# B&R Automation Studio project Nikhil_5_Axes
Automation Studio 4.12.2.93; technology packages: mapp 5.24.1, mappCockpit 5.24.1, mappMotion 5.31.0, mappView 5.24.0, mappVision 5.24.0

## Configuration X20CP0484

CPU X20CP0484-1, AutomationRuntime B4.93, Build 4.1.2, Safety 0.0, Vc V4.72.6

### Task classes (Cpu.sw)
```
Cyclic#1 (cycle 4000 us, tolerance 0 us):
  Motion_Con <- Motion_Control.prg
DataObjects: McAcpSys
NcDataObjects: McDriveLog
Binaries: visionUnit, mvLoader, arcoal, arflatprv, arsvcreg, mcprofgen, TCLang, TCData, McPathXT, McAcpSim, mCoWebSc, FWRules, McAcpDrv, udbdef, OpcUaSrv, McMechSys, Role, Config_3, arconfig, Settings, User, asfw, ashwd, Config_1, ashwac, TraceConfi, TC, sysconf, Config_4, Config, Hierarchy, iomap, Config_2, Config_5
Libraries: McBase, MpRobotics, McAxGroup, MpBase, McPathGen, McAxis, McProgInt, McAcpAx, CoTrace, AsZip, FileIO, runtime, ViBase, AsARCfg, powerlnk, AsEPL, AsIO, sys_lib, astime, McStpAx, DataObj, MpAxis, McTrkPath, MpPick, AsOpcUac, AsOpcUas, asarlog, asmem, asieccon, brsystem, asarprof, arssl, asioacc
```

### Hardware
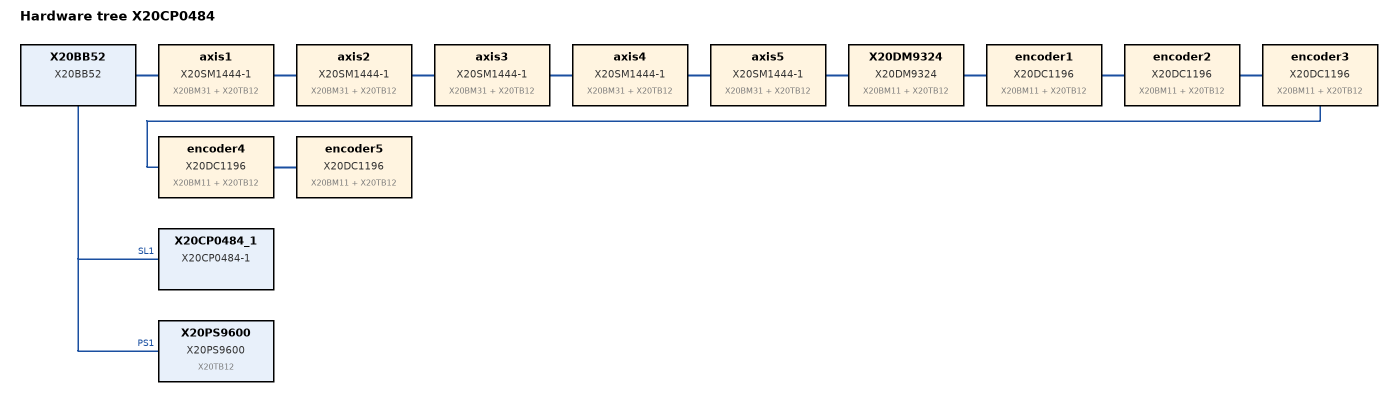
```
X20BB52 : X20BB52 v1.2.0.0
X20BM11 : X20BM11 v1.1.0.0  [X2X1 -> X20BM31d.X2X2]
X20BM11a : X20BM11 v1.1.0.0  [X2X1 -> X20BM11.X2X2]
X20BM11b : X20BM11 v1.1.0.0  [X2X1 -> X20BM11a.X2X2]
X20BM11c : X20BM11 v1.1.0.0  [X2X1 -> X20BM11b.X2X2]
X20BM11d : X20BM11 v1.1.0.0  [X2X1 -> X20BM11c.X2X2]
X20BM11e : X20BM11 v1.1.0.0  [X2X1 -> X20BM11d.X2X2]
X20BM31 : X20BM31 v1.1.0.0  [X2X1 -> X20BB52.IF6]
X20BM31a : X20BM31 v1.1.0.0  [X2X1 -> X20BM31.X2X2]
X20BM31b : X20BM31 v1.1.0.0  [X2X1 -> X20BM31a.X2X2]
X20BM31c : X20BM31 v1.1.0.0  [X2X1 -> X20BM31b.X2X2]
X20BM31d : X20BM31 v1.1.0.0  [X2X1 -> X20BM31c.X2X2]
X20CP0484_1 : X20CP0484-1 v1.4.0.0  [SL -> X20BB52.SL1]
  Connector IF2:
    ActivateDevice = 1
    Mode = Manual
    InternetAddress = 169.254.137.11
    SubnetMask = 255.255.255.0
    InaNodeNumber = 1
    ActivateSnmp = 2
  ConfigurationID = Nikhil_5_Axes
  AutomaticTransferOfUserfiles = on
  MotionLoggerSize = 2048000
  TimerDeviceType = EPLX2X
  TimerDevice = X20BB52.IF6
  TaskClassIdleTime = 4000
  Cyclic1Duration = 4000
  Cyclic1Tolerance = 0
  Cyclic2Duration = 20000
  Cyclic2Tolerance = 20000
  Cyclic3Duration = 48000
  Cyclic3Tolerance = 48000
  Cyclic4Duration = 100000
  Cyclic4Tolerance = 100000
  Cyclic5Duration = 200000
  Cyclic5Tolerance = 200000
  Cyclic6Duration = 500000
  Cyclic6Tolerance = 500000
  Cyclic7Duration = 1000000
  Cyclic7Tolerance = 1000000
  Cyclic8Duration = 8000
  Cyclic8Tolerance = 30000000
  FileDevice1
  FileDeviceName1 = Simulation
  FileDevicePath1 = Z:\Nikhil\Project_5_Axes\Nikhil_test\Logical\CNC_PrgDir
  FileDevice2
  FileDeviceName2 = CNC_PrgDir
  FileDevicePath2 = F:\
  FileDevice3
  FileDeviceName3 = SceneViewer
  FileDevicePath3 = Z:\Nikhil\Project_5_Axes\Nikhil_test\Logical\SceneViewer
  ActivateDns = 1
  DnsDefaultDomain = br-automation.co.at
  FtpUser1
  FtpUsername1 = user
  FtpUserPassword1 = soUu8fSmbl9vOUGFZLohNxYIHTvfYbNb9FbAKhZ+648=
  FtpUserSalt1 = plFIy1g6
  FTPAccessRight1 = 0
  FTPdevice1 = ALL
  ActivateDtmServer = 1
  ActivateOpcUa = 1
  OpcUaPort = 48400
  OpcUa_AuthenticationSecurityPolicy_EnableNone = 1
  OpcUa_AuthenticationSecurityPolicy_EnableBasic128Rsa15 = 1
  OpcUa_Security_AdminRole = Administrators
  OpcUa_Security_EngineerRole = Everyone
  OpcUa_Security_ObserverRole = Everyone
  OpcUaInformationModels_PV_Version = 2
  OpcUaInformationModel_Facet = 0
  OpcUaInformationModel_TypeInformation = 0
  OpcUaInformationModel_BaseObjectTypeForStructures = 0
X20DM9324 : X20DM9324 v1.2.0.0  [SS1 -> X20TB12f.SS; SL -> X20BM11.SL1]
X20PS9600 : X20PS9600 v1.6.0.0  [PS -> X20BB52.PS1; SS1 -> X20TB12.SS]
X20TB12 : X20TB12 v1.0.0.0
X20TB12a : X20TB12 v1.0.0.0
X20TB12b : X20TB12 v1.0.0.0
X20TB12c : X20TB12 v1.0.0.0
X20TB12d : X20TB12 v1.0.0.0
X20TB12e : X20TB12 v1.0.0.0
X20TB12f : X20TB12 v1.0.0.0
X20TB12g : X20TB12 v1.0.0.0
X20TB12h : X20TB12 v1.0.0.0
X20TB12i : X20TB12 v1.0.0.0
X20TB12j : X20TB12 v1.0.0.0
X20TB12k : X20TB12 v1.0.0.0
axis1 : X20SM1444-1 v1.2.0.0  [SS1 -> X20TB12a.SS; SL -> X20BM31.SL1]
  FunctionModel/DriveConfiguration/Module:
    ActivateModuleSimulationOnPLC = Off
  FunctionModel/DriveConfiguration:
    ModuleParameters = StepperParameters
  FunctionModel/DriveConfiguration/ModuleParameters:
    McStepperTypeID = X20Config
    EncoderType = IncrementalDiff
    ReferencePulse = yes
    RatedCurrent = 5.0
    MaximumCurrent = 10.0
    AxesNumber = 1
    FullStepThreshold = 1
    StallDetection = 2
    SmartCurrentControl = 1
    BrakeOutput = 0
    NumberOfDigitalInputs = 3
    NumberOfTriggers = 1
  FunctionModel/DriveConfiguration/Channel[1]/RealAxis:
    AxisReference = gAxisQ1
  FunctionModel/DriveConfiguration/Channel[1]/RealAxis/MechanicalElements/Gearbox:
    InputIsReadOnly = 0
    Input = 48
    OutputIsReadOnly = 0
    Output = 1
  FunctionModel/DriveConfiguration/Channel[1]/RealAxis/MechanicalElements/RotaryToLinearTransformation:
    ReferenceDistanceIsReadOnly = 0
    ReferenceDistance = 1
  FunctionModel/DriveConfiguration/Channel[1]/RealAxis/Motor:
    SteppingAngle = 1.8
  FunctionModel/DriveConfiguration/Channel[1]/RealAxis:
    EncoderLink = OneEncoder
  FunctionModel/DriveConfiguration/Channel[1]/RealAxis/EncoderLink:
    PositionEncoder = External
  FunctionModel/DriveConfiguration/Channel[1]/RealAxis/EncoderLink/PositionEncoder:
    LinesPerRevolution = 2000
    PositionType = Incremental
  FunctionModel/DriveConfiguration/Channel[1]/RealAxis/EncoderLink/PositionEncoder/PositionSource:
    ChannelMapping = %ID.IF6.ST7.Encoder01
  FunctionModel/DriveConfiguration/Channel[1]/RealAxis/EncoderLink/PositionEncoder/ValidityCheck:
    ModuleOk = IOChannel
  FunctionModel/DriveConfiguration/Channel[1]/RealAxis/EncoderLink/PositionEncoder/ValidityCheck/ModuleOk:
    ChannelMapping = %IX.IF6.ST7.ModuleOk
  FunctionModel/DriveConfiguration/Channel[1]/RealAxis/EncoderLink/PositionEncoder/ValidityCheck:
    StaleData = IOChannel
  FunctionModel/DriveConfiguration/Channel[1]/RealAxis/EncoderLink/PositionEncoder/ValidityCheck/StaleData:
    ChannelMapping = %IX.IF6.ST7.StaleData
  FunctionModel/DriveConfiguration/Channel[1]/RealAxis/EncoderLink/PositionEncoder:
    ReferencePulse = NotUsed
  FunctionModel/DriveConfiguration/Channel[1]/RealAxis/EncoderLink/PositionEncoder/PositionFilter:
    PositionFilterTimeConstant = 0.0
    ExtrapolationTime = 0.0
  FunctionModel/DriveConfiguration/Channel[1]/RealAxis/Controller:
    ModeIsReadOnly = 0
    Mode = CurrentController
  FunctionModel/DriveConfiguration/Channel[1]/RealAxis/Controller/Mode/Current:
    StandstillCurrent = 1
    ConstantSpeedCurrent = 4
    SpeedChangeCurrent = 4.2
    FullStepThreshold = 0.0
    MotorSettlingTime = 1
    DelayedCurrentSwitchOff = 1
  FunctionModel/DriveConfiguration/Channel[1]/RealAxis/Homing:
    Mode = AbsoluteSwitch
  FunctionModel/DriveConfiguration/Channel[1]/RealAxis/Homing/Mode:
    Position = 0.0
    StartVelocity = 5.0
    HomingVelocity = 2
    Acceleration = 50.0
    SwitchEdge = Positive
    HomingDirection = Positive
    KeepDirection = No
    ReferencePulse = NotUsed
  FunctionModel/DriveConfiguration/Channel[1]/RealAxis/Homing:
    RestorePositionVariable = 
    ClearPositionError = No
  FunctionModel/DriveConfiguration/Channel[1]/RealAxis/StopReaction:
    DriveError = DecelerationLimit
  FunctionModel/DriveConfiguration/Channel[1]/RealAxis/MovementErrorLimits:
    PositionError = 1000
    StallguardConfiguration = NotUsed
  FunctionModel/DriveConfiguration/Channel[1]/RealAxis:
    JerkFilter = NotUsed
    ZeroVibrationFilter = NotUsed
  FunctionModel/DriveConfiguration/Channel[1]/RealAxis/DigitalInputs/HomingSwitch:
    Source = IOChannel
  FunctionModel/DriveConfiguration/Channel[1]/RealAxis/DigitalInputs/HomingSwitch/Source:
    ChannelMapping = %IX.IF6.ST6.DigitalInput01
  FunctionModel/DriveConfiguration/Channel[1]/RealAxis/DigitalInputs/HomingSwitch:
    Level = Low
  FunctionModel/DriveConfiguration/Channel[1]/RealAxis/DigitalInputs/PositiveLimitSwitch:
    Source = NotUsed
    Level = High
  FunctionModel/DriveConfiguration/Channel[1]/RealAxis/DigitalInputs/NegativeLimitSwitch:
    Source = NotUsed
    Level = High
  FunctionModel/DriveConfiguration/Channel[1]/RealAxis/DigitalInputs/Trigger1:
    Source = NotUsed
    Level = High
  FunctionModel/DriveConfiguration/Channel[1]/RealAxis/DigitalInputs/Trigger2:
    Source = NotUsed
    Level = High
  FunctionModel/DriveConfiguration/Channel[1]/RealAxis/DigitalInputs/Quickstop:
    Input = NotUsed
  FunctionModel/DriveConfiguration/Channel[1]/RealAxis/DigitalOutputs:
    BrakeControl = NotUsed
  FunctionModel/DriveConfiguration/Channel[1]/RealAxis/Simulation:
    LoadSimulationMode = NotUsed
axis2 : X20SM1444-1 v1.2.0.0  [SS1 -> X20TB12b.SS; SL -> X20BM31a.SL1]
  FunctionModel/DriveConfiguration/Module:
    ActivateModuleSimulationOnPLC = Off
  FunctionModel/DriveConfiguration:
    ModuleParameters = StepperParameters
  FunctionModel/DriveConfiguration/ModuleParameters:
    McStepperTypeID = X20Config
    EncoderType = IncrementalDiff
    ReferencePulse = yes
    RatedCurrent = 5.0
    MaximumCurrent = 10.0
    AxesNumber = 1
    FullStepThreshold = 1
    StallDetection = 2
    SmartCurrentControl = 1
    BrakeOutput = 0
    NumberOfDigitalInputs = 3
    NumberOfTriggers = 1
  FunctionModel/DriveConfiguration/Channel[1]/RealAxis:
    AxisReference = gAxisQ2
  FunctionModel/DriveConfiguration/Channel[1]/RealAxis/MechanicalElements/Gearbox:
    InputIsReadOnly = 0
    Input = 48
    OutputIsReadOnly = 0
    Output = 1
  FunctionModel/DriveConfiguration/Channel[1]/RealAxis/MechanicalElements/RotaryToLinearTransformation:
    ReferenceDistanceIsReadOnly = 0
    ReferenceDistance = 1
  FunctionModel/DriveConfiguration/Channel[1]/RealAxis/Motor:
    SteppingAngle = 1.8
  FunctionModel/DriveConfiguration/Channel[1]/RealAxis:
    EncoderLink = OneEncoder
  FunctionModel/DriveConfiguration/Channel[1]/RealAxis/EncoderLink:
    PositionEncoder = External
  FunctionModel/DriveConfiguration/Channel[1]/RealAxis/EncoderLink/PositionEncoder:
    LinesPerRevolution = 2000
    PositionType = Incremental
  FunctionModel/DriveConfiguration/Channel[1]/RealAxis/EncoderLink/PositionEncoder/PositionSource:
    ChannelMapping = %ID.IF6.ST8.Encoder01
  FunctionModel/DriveConfiguration/Channel[1]/RealAxis/EncoderLink/PositionEncoder/ValidityCheck:
    ModuleOk = IOChannel
  FunctionModel/DriveConfiguration/Channel[1]/RealAxis/EncoderLink/PositionEncoder/ValidityCheck/ModuleOk:
    ChannelMapping = %IX.IF6.ST8.ModuleOk
  FunctionModel/DriveConfiguration/Channel[1]/RealAxis/EncoderLink/PositionEncoder/ValidityCheck:
    StaleData = IOChannel
  FunctionModel/DriveConfiguration/Channel[1]/RealAxis/EncoderLink/PositionEncoder/ValidityCheck/StaleData:
    ChannelMapping = %IX.IF6.ST8.StaleData
  FunctionModel/DriveConfiguration/Channel[1]/RealAxis/EncoderLink/PositionEncoder:
    ReferencePulse = NotUsed
  FunctionModel/DriveConfiguration/Channel[1]/RealAxis/EncoderLink/PositionEncoder/PositionFilter:
    PositionFilterTimeConstant = 0.0
    ExtrapolationTime = 0.0
  FunctionModel/DriveConfiguration/Channel[1]/RealAxis/Controller:
    ModeIsReadOnly = 0
    Mode = CurrentController
  FunctionModel/DriveConfiguration/Channel[1]/RealAxis/Controller/Mode/Current:
    StandstillCurrent = 1
    ConstantSpeedCurrent = 4.2
    SpeedChangeCurrent = 4.2
    FullStepThreshold = 0.0
    MotorSettlingTime = 1
    DelayedCurrentSwitchOff = 1
  FunctionModel/DriveConfiguration/Channel[1]/RealAxis/Homing:
    Mode = AbsoluteSwitch
  FunctionModel/DriveConfiguration/Channel[1]/RealAxis/Homing/Mode:
    Position = -10
    StartVelocity = 5.0
    HomingVelocity = 2
    Acceleration = 50.0
    SwitchEdge = Negative
    HomingDirection = Negative
    KeepDirection = No
    ReferencePulse = NotUsed
  FunctionModel/DriveConfiguration/Channel[1]/RealAxis/Homing:
    RestorePositionVariable = 
    ClearPositionError = No
  FunctionModel/DriveConfiguration/Channel[1]/RealAxis/StopReaction:
    DriveError = DecelerationLimit
  FunctionModel/DriveConfiguration/Channel[1]/RealAxis/MovementErrorLimits:
    PositionError = 1000
    StallguardConfiguration = NotUsed
  FunctionModel/DriveConfiguration/Channel[1]/RealAxis:
    JerkFilter = NotUsed
    ZeroVibrationFilter = NotUsed
  FunctionModel/DriveConfiguration/Channel[1]/RealAxis/DigitalInputs/HomingSwitch:
    Source = IOChannel
  FunctionModel/DriveConfiguration/Channel[1]/RealAxis/DigitalInputs/HomingSwitch/Source:
    ChannelMapping = %IX.IF6.ST6.DigitalInput02
  FunctionModel/DriveConfiguration/Channel[1]/RealAxis/DigitalInputs/HomingSwitch:
    Level = Low
  FunctionModel/DriveConfiguration/Channel[1]/RealAxis/DigitalInputs/PositiveLimitSwitch:
    Source = NotUsed
    Level = High
  FunctionModel/DriveConfiguration/Channel[1]/RealAxis/DigitalInputs/NegativeLimitSwitch:
    Source = NotUsed
    Level = High
  FunctionModel/DriveConfiguration/Channel[1]/RealAxis/DigitalInputs/Trigger1:
    Source = NotUsed
    Level = High
  FunctionModel/DriveConfiguration/Channel[1]/RealAxis/DigitalInputs/Trigger2:
    Source = NotUsed
    Level = High
  FunctionModel/DriveConfiguration/Channel[1]/RealAxis/DigitalInputs/Quickstop:
    Input = NotUsed
  FunctionModel/DriveConfiguration/Channel[1]/RealAxis/DigitalOutputs:
    BrakeControl = NotUsed
  FunctionModel/DriveConfiguration/Channel[1]/RealAxis/Simulation:
    LoadSimulationMode = NotUsed
axis3 : X20SM1444-1 v1.2.0.0  [SS1 -> X20TB12c.SS; SL -> X20BM31b.SL1]
  FunctionModel/DriveConfiguration/Module:
    ActivateModuleSimulationOnPLC = Off
  FunctionModel/DriveConfiguration:
    ModuleParameters = StepperParameters
  FunctionModel/DriveConfiguration/ModuleParameters:
    McStepperTypeID = X20Config
    EncoderType = IncrementalDiff
    ReferencePulse = yes
    RatedCurrent = 5.0
    MaximumCurrent = 10.0
    AxesNumber = 1
    FullStepThreshold = 1
    StallDetection = 2
    SmartCurrentControl = 1
    BrakeOutput = 0
    NumberOfDigitalInputs = 3
    NumberOfTriggers = 1
  FunctionModel/DriveConfiguration/Channel[1]/RealAxis:
    AxisReference = gAxisQ3
  FunctionModel/DriveConfiguration/Channel[1]/RealAxis/MechanicalElements/Gearbox:
    InputIsReadOnly = 0
    Input = 50
    OutputIsReadOnly = 0
    Output = 1
  FunctionModel/DriveConfiguration/Channel[1]/RealAxis/MechanicalElements/RotaryToLinearTransformation:
    ReferenceDistanceIsReadOnly = 0
    ReferenceDistance = 1
  FunctionModel/DriveConfiguration/Channel[1]/RealAxis/Motor:
    SteppingAngle = 1.8
  FunctionModel/DriveConfiguration/Channel[1]/RealAxis:
    EncoderLink = OneEncoder
  FunctionModel/DriveConfiguration/Channel[1]/RealAxis/EncoderLink:
    PositionEncoder = External
  FunctionModel/DriveConfiguration/Channel[1]/RealAxis/EncoderLink/PositionEncoder:
    LinesPerRevolution = 2000
    PositionType = Incremental
  FunctionModel/DriveConfiguration/Channel[1]/RealAxis/EncoderLink/PositionEncoder/PositionSource:
    ChannelMapping = %ID.IF6.ST9.Encoder01
  FunctionModel/DriveConfiguration/Channel[1]/RealAxis/EncoderLink/PositionEncoder/ValidityCheck:
    ModuleOk = IOChannel
  FunctionModel/DriveConfiguration/Channel[1]/RealAxis/EncoderLink/PositionEncoder/ValidityCheck/ModuleOk:
    ChannelMapping = %IX.IF6.ST9.ModuleOk
  FunctionModel/DriveConfiguration/Channel[1]/RealAxis/EncoderLink/PositionEncoder/ValidityCheck:
    StaleData = IOChannel
  FunctionModel/DriveConfiguration/Channel[1]/RealAxis/EncoderLink/PositionEncoder/ValidityCheck/StaleData:
    ChannelMapping = %IX.IF6.ST9.StaleData
  FunctionModel/DriveConfiguration/Channel[1]/RealAxis/EncoderLink/PositionEncoder:
    ReferencePulse = NotUsed
  FunctionModel/DriveConfiguration/Channel[1]/RealAxis/EncoderLink/PositionEncoder/PositionFilter:
    PositionFilterTimeConstant = 0.0
    ExtrapolationTime = 0.0
  FunctionModel/DriveConfiguration/Channel[1]/RealAxis/Controller:
    ModeIsReadOnly = 0
    Mode = CurrentController
  FunctionModel/DriveConfiguration/Channel[1]/RealAxis/Controller/Mode/Current:
    StandstillCurrent = 1
    ConstantSpeedCurrent = 4.2
    SpeedChangeCurrent = 4.2
    FullStepThreshold = 0.0
    MotorSettlingTime = 1
    DelayedCurrentSwitchOff = 1
  FunctionModel/DriveConfiguration/Channel[1]/RealAxis/Homing:
    Mode = AbsoluteSwitch
  FunctionModel/DriveConfiguration/Channel[1]/RealAxis/Homing/Mode:
    Position = 10
    StartVelocity = 5.0
    HomingVelocity = 2
    Acceleration = 50.0
    SwitchEdge = Negative
    HomingDirection = Negative
    KeepDirection = No
    ReferencePulse = NotUsed
  FunctionModel/DriveConfiguration/Channel[1]/RealAxis/Homing:
    RestorePositionVariable = 
    ClearPositionError = No
  FunctionModel/DriveConfiguration/Channel[1]/RealAxis/StopReaction:
    DriveError = DecelerationLimit
  FunctionModel/DriveConfiguration/Channel[1]/RealAxis/MovementErrorLimits:
    PositionError = 1000
    StallguardConfiguration = NotUsed
  FunctionModel/DriveConfiguration/Channel[1]/RealAxis:
    JerkFilter = NotUsed
    ZeroVibrationFilter = NotUsed
  FunctionModel/DriveConfiguration/Channel[1]/RealAxis/DigitalInputs/HomingSwitch:
    Source = IOChannel
  FunctionModel/DriveConfiguration/Channel[1]/RealAxis/DigitalInputs/HomingSwitch/Source:
    ChannelMapping = %IX.IF6.ST6.DigitalInput03
  FunctionModel/DriveConfiguration/Channel[1]/RealAxis/DigitalInputs/HomingSwitch:
    Level = Low
  FunctionModel/DriveConfiguration/Channel[1]/RealAxis/DigitalInputs/PositiveLimitSwitch:
    Source = NotUsed
    Level = High
  FunctionModel/DriveConfiguration/Channel[1]/RealAxis/DigitalInputs/NegativeLimitSwitch:
    Source = NotUsed
    Level = High
  FunctionModel/DriveConfiguration/Channel[1]/RealAxis/DigitalInputs/Trigger1:
    Source = NotUsed
    Level = High
  FunctionModel/DriveConfiguration/Channel[1]/RealAxis/DigitalInputs/Trigger2:
    Source = NotUsed
    Level = High
  FunctionModel/DriveConfiguration/Channel[1]/RealAxis/DigitalInputs/Quickstop:
    Input = NotUsed
  FunctionModel/DriveConfiguration/Channel[1]/RealAxis/DigitalOutputs:
    BrakeControl = NotUsed
  FunctionModel/DriveConfiguration/Channel[1]/RealAxis/Simulation:
    LoadSimulationMode = NotUsed
axis4 : X20SM1444-1 v1.2.0.0  [SS1 -> X20TB12d.SS; SL -> X20BM31c.SL1]
  FunctionModel/DriveConfiguration/Module:
    ActivateModuleSimulationOnPLC = Off
  FunctionModel/DriveConfiguration:
    ModuleParameters = StepperParameters
  FunctionModel/DriveConfiguration/ModuleParameters:
    McStepperTypeID = X20Config
    EncoderType = IncrementalDiff
    ReferencePulse = yes
    RatedCurrent = 5.0
    MaximumCurrent = 10.0
    AxesNumber = 1
    FullStepThreshold = 1
    StallDetection = 2
    SmartCurrentControl = 1
    BrakeOutput = 0
    NumberOfDigitalInputs = 3
    NumberOfTriggers = 1
  FunctionModel/DriveConfiguration/Channel[1]/RealAxis:
    AxisReference = gAxisQ4
  FunctionModel/DriveConfiguration/Channel[1]/RealAxis/MechanicalElements/Gearbox:
    InputIsReadOnly = 0
    Input = 40
    OutputIsReadOnly = 0
    Output = 1
  FunctionModel/DriveConfiguration/Channel[1]/RealAxis/MechanicalElements/RotaryToLinearTransformation:
    ReferenceDistanceIsReadOnly = 0
    ReferenceDistance = 1
  FunctionModel/DriveConfiguration/Channel[1]/RealAxis/Motor:
    SteppingAngle = 1.8
  FunctionModel/DriveConfiguration/Channel[1]/RealAxis:
    EncoderLink = OneEncoder
  FunctionModel/DriveConfiguration/Channel[1]/RealAxis/EncoderLink:
    PositionEncoder = External
  FunctionModel/DriveConfiguration/Channel[1]/RealAxis/EncoderLink/PositionEncoder:
    LinesPerRevolution = 2000
    PositionType = Incremental
  FunctionModel/DriveConfiguration/Channel[1]/RealAxis/EncoderLink/PositionEncoder/PositionSource:
    ChannelMapping = %ID.IF6.ST10.Encoder01
  FunctionModel/DriveConfiguration/Channel[1]/RealAxis/EncoderLink/PositionEncoder/ValidityCheck:
    ModuleOk = IOChannel
  FunctionModel/DriveConfiguration/Channel[1]/RealAxis/EncoderLink/PositionEncoder/ValidityCheck/ModuleOk:
    ChannelMapping = %IX.IF6.ST10.ModuleOk
  FunctionModel/DriveConfiguration/Channel[1]/RealAxis/EncoderLink/PositionEncoder/ValidityCheck:
    StaleData = IOChannel
  FunctionModel/DriveConfiguration/Channel[1]/RealAxis/EncoderLink/PositionEncoder/ValidityCheck/StaleData:
    ChannelMapping = %IX.IF6.ST10.StaleData
  FunctionModel/DriveConfiguration/Channel[1]/RealAxis/EncoderLink/PositionEncoder:
    ReferencePulse = NotUsed
  FunctionModel/DriveConfiguration/Channel[1]/RealAxis/EncoderLink/PositionEncoder/PositionFilter:
    PositionFilterTimeConstant = 0.0
    ExtrapolationTime = 0.0
  FunctionModel/DriveConfiguration/Channel[1]/RealAxis/Controller:
    ModeIsReadOnly = 0
    Mode = CurrentController
  FunctionModel/DriveConfiguration/Channel[1]/RealAxis/Controller/Mode/Current:
    StandstillCurrent = 0.6
    ConstantSpeedCurrent = 1.8
    SpeedChangeCurrent = 1.8
    FullStepThreshold = 0.0
    MotorSettlingTime = 1
    DelayedCurrentSwitchOff = 1
  FunctionModel/DriveConfiguration/Channel[1]/RealAxis/Homing:
    Mode = AbsoluteSwitch
  FunctionModel/DriveConfiguration/Channel[1]/RealAxis/Homing/Mode:
    Position = -10
    StartVelocity = 5.0
    HomingVelocity = 2
    Acceleration = 50.0
    SwitchEdge = Positive
    HomingDirection = Positive
    KeepDirection = No
    ReferencePulse = NotUsed
  FunctionModel/DriveConfiguration/Channel[1]/RealAxis/Homing:
    RestorePositionVariable = 
    ClearPositionError = No
  FunctionModel/DriveConfiguration/Channel[1]/RealAxis/StopReaction:
    DriveError = DecelerationLimit
  FunctionModel/DriveConfiguration/Channel[1]/RealAxis/MovementErrorLimits:
    PositionError = 1000
    StallguardConfiguration = NotUsed
  FunctionModel/DriveConfiguration/Channel[1]/RealAxis:
    JerkFilter = NotUsed
    ZeroVibrationFilter = NotUsed
  FunctionModel/DriveConfiguration/Channel[1]/RealAxis/DigitalInputs/HomingSwitch:
    Source = IOChannel
  FunctionModel/DriveConfiguration/Channel[1]/RealAxis/DigitalInputs/HomingSwitch/Source:
    ChannelMapping = %IX.IF6.ST6.DigitalInput04
  FunctionModel/DriveConfiguration/Channel[1]/RealAxis/DigitalInputs/HomingSwitch:
    Level = Low
  FunctionModel/DriveConfiguration/Channel[1]/RealAxis/DigitalInputs/PositiveLimitSwitch:
    Source = NotUsed
    Level = High
  FunctionModel/DriveConfiguration/Channel[1]/RealAxis/DigitalInputs/NegativeLimitSwitch:
    Source = NotUsed
    Level = High
  FunctionModel/DriveConfiguration/Channel[1]/RealAxis/DigitalInputs/Trigger1:
    Source = NotUsed
    Level = High
  FunctionModel/DriveConfiguration/Channel[1]/RealAxis/DigitalInputs/Trigger2:
    Source = NotUsed
    Level = High
  FunctionModel/DriveConfiguration/Channel[1]/RealAxis/DigitalInputs/Quickstop:
    Input = NotUsed
  FunctionModel/DriveConfiguration/Channel[1]/RealAxis/DigitalOutputs:
    BrakeControl = NotUsed
  FunctionModel/DriveConfiguration/Channel[1]/RealAxis/Simulation:
    LoadSimulationMode = NotUsed
axis5 : X20SM1444-1 v1.2.0.0  [SS1 -> X20TB12e.SS; SL -> X20BM31d.SL1]
  FunctionModel/DriveConfiguration/Module:
    ActivateModuleSimulationOnPLC = Off
  FunctionModel/DriveConfiguration:
    ModuleParameters = StepperParameters
  FunctionModel/DriveConfiguration/ModuleParameters:
    McStepperTypeID = X20Config
    EncoderType = IncrementalDiff
    ReferencePulse = yes
    RatedCurrent = 5.0
    MaximumCurrent = 10.0
    AxesNumber = 1
    FullStepThreshold = 1
    StallDetection = 2
    SmartCurrentControl = 1
    BrakeOutput = 0
    NumberOfDigitalInputs = 3
    NumberOfTriggers = 1
  FunctionModel/DriveConfiguration/Channel[1]/RealAxis:
    AxisReference = gAxisQ5
  FunctionModel/DriveConfiguration/Channel[1]/RealAxis/MechanicalElements/Gearbox:
    InputIsReadOnly = 0
    Input = 28
    OutputIsReadOnly = 0
    Output = 1
  FunctionModel/DriveConfiguration/Channel[1]/RealAxis/MechanicalElements/RotaryToLinearTransformation:
    ReferenceDistanceIsReadOnly = 0
    ReferenceDistance = 1
  FunctionModel/DriveConfiguration/Channel[1]/RealAxis/Motor:
    SteppingAngle = 1.8
  FunctionModel/DriveConfiguration/Channel[1]/RealAxis:
    EncoderLink = OneEncoder
  FunctionModel/DriveConfiguration/Channel[1]/RealAxis/EncoderLink:
    PositionEncoder = External
  FunctionModel/DriveConfiguration/Channel[1]/RealAxis/EncoderLink/PositionEncoder:
    LinesPerRevolution = 2000
    PositionType = Incremental
  FunctionModel/DriveConfiguration/Channel[1]/RealAxis/EncoderLink/PositionEncoder/PositionSource:
    ChannelMapping = %ID.IF6.ST11.Encoder01
  FunctionModel/DriveConfiguration/Channel[1]/RealAxis/EncoderLink/PositionEncoder/ValidityCheck:
    ModuleOk = IOChannel
  FunctionModel/DriveConfiguration/Channel[1]/RealAxis/EncoderLink/PositionEncoder/ValidityCheck/ModuleOk:
    ChannelMapping = %IX.IF6.ST11.ModuleOk
  FunctionModel/DriveConfiguration/Channel[1]/RealAxis/EncoderLink/PositionEncoder/ValidityCheck:
    StaleData = IOChannel
  FunctionModel/DriveConfiguration/Channel[1]/RealAxis/EncoderLink/PositionEncoder/ValidityCheck/StaleData:
    ChannelMapping = %IX.IF6.ST11.StaleData
  FunctionModel/DriveConfiguration/Channel[1]/RealAxis/EncoderLink/PositionEncoder:
    ReferencePulse = NotUsed
  FunctionModel/DriveConfiguration/Channel[1]/RealAxis/EncoderLink/PositionEncoder/PositionFilter:
    PositionFilterTimeConstant = 0.0
    ExtrapolationTime = 0.0
  FunctionModel/DriveConfiguration/Channel[1]/RealAxis/Controller:
    ModeIsReadOnly = 0
    Mode = CurrentController
  FunctionModel/DriveConfiguration/Channel[1]/RealAxis/Controller/Mode/Current:
    StandstillCurrent = 0.2
    ConstantSpeedCurrent = 1.8
    SpeedChangeCurrent = 1.8
    FullStepThreshold = 0.0
    MotorSettlingTime = 1
    DelayedCurrentSwitchOff = 1
  FunctionModel/DriveConfiguration/Channel[1]/RealAxis/Homing:
    Mode = AbsoluteSwitch
  FunctionModel/DriveConfiguration/Channel[1]/RealAxis/Homing/Mode:
    Position = -10
    StartVelocity = 5.0
    HomingVelocity = 2
    Acceleration = 50.0
    SwitchEdge = Positive
    HomingDirection = Negative
    KeepDirection = No
    ReferencePulse = NotUsed
  FunctionModel/DriveConfiguration/Channel[1]/RealAxis/Homing:
    RestorePositionVariable = 
    ClearPositionError = No
  FunctionModel/DriveConfiguration/Channel[1]/RealAxis/StopReaction:
    DriveError = DecelerationLimit
  FunctionModel/DriveConfiguration/Channel[1]/RealAxis/MovementErrorLimits:
    PositionError = 1000
    StallguardConfiguration = NotUsed
  FunctionModel/DriveConfiguration/Channel[1]/RealAxis:
    JerkFilter = NotUsed
    ZeroVibrationFilter = NotUsed
  FunctionModel/DriveConfiguration/Channel[1]/RealAxis/DigitalInputs/HomingSwitch:
    Source = IOChannel
  FunctionModel/DriveConfiguration/Channel[1]/RealAxis/DigitalInputs/HomingSwitch/Source:
    ChannelMapping = %IX.IF6.ST6.DigitalInput05
  FunctionModel/DriveConfiguration/Channel[1]/RealAxis/DigitalInputs/HomingSwitch:
    Level = Low
  FunctionModel/DriveConfiguration/Channel[1]/RealAxis/DigitalInputs/PositiveLimitSwitch:
    Source = NotUsed
    Level = High
  FunctionModel/DriveConfiguration/Channel[1]/RealAxis/DigitalInputs/NegativeLimitSwitch:
    Source = NotUsed
    Level = High
  FunctionModel/DriveConfiguration/Channel[1]/RealAxis/DigitalInputs/Trigger1:
    Source = NotUsed
    Level = High
  FunctionModel/DriveConfiguration/Channel[1]/RealAxis/DigitalInputs/Trigger2:
    Source = NotUsed
    Level = High
  FunctionModel/DriveConfiguration/Channel[1]/RealAxis/DigitalInputs/Quickstop:
    Input = NotUsed
  FunctionModel/DriveConfiguration/Channel[1]/RealAxis/DigitalOutputs:
    BrakeControl = NotUsed
  FunctionModel/DriveConfiguration/Channel[1]/RealAxis/Simulation:
    LoadSimulationMode = NotUsed
encoder1 : X20DC1196 v1.4.0.0  [SS1 -> X20TB12g.SS; SL -> X20BM11a.SL1]
  FunctionModel = FunctionModel001
encoder2 : X20DC1196 v1.4.0.0  [SS1 -> X20TB12h.SS; SL -> X20BM11b.SL1]
  FunctionModel = FunctionModel001
encoder3 : X20DC1196 v1.4.0.0  [SS1 -> X20TB12i.SS; SL -> X20BM11c.SL1]
  FunctionModel = FunctionModel001
encoder4 : X20DC1196 v1.4.0.0  [SS1 -> X20TB12j.SS; SL -> X20BM11d.SL1]
  FunctionModel = FunctionModel001
encoder5 : X20DC1196 v1.4.0.0  [SS1 -> X20TB12k.SS; SL -> X20BM11e.SL1]
  FunctionModel = FunctionModel001
```

### IoMap.iom - X20CP0484_1/IoMap.iom
```iecst
VAR_CONFIG
	::gEStop_OK AT %IX."X20DM9324".DigitalInput06;
	::SM_Module_TriggerVars.Axis1 AT %IX."X20DM9324".DigitalInput01;
	::SM_Module_TriggerVars.Axis2 AT %IX."X20DM9324".DigitalInput02;
	::SM_Module_TriggerVars.Axis3 AT %IX."X20DM9324".DigitalInput03;
	::SM_Module_TriggerVars.Axis4 AT %IX."X20DM9324".DigitalInput04;
	::SM_Module_TriggerVars.Axis5 AT %IX."X20DM9324".DigitalInput05;
	::Motion_Con:gGripperOpen AT %QX."X20DM9324".DigitalOutput01;
	::Motion_Con:gGripperClose AT %QX."X20DM9324".DigitalOutput02;
END_VAR
```

### Config_1.axesgroup - X20CP0484_1/mappMotion/5AxesRoboarmA/Config_1.axesgroup
```
Element g5AxRobA (Type=axesgroup)
  Type = PathGenAxesGroup
    ProcessingTaskClass = 1
    License = 1
    PhysicalAxes:
      JointAxes:
        JointAxis[1]:
          Name = Q1
          AxisRef = gAxisQ1
        JointAxis[2]:
          Name = Q2
          AxisRef = gAxisQ2
        JointAxis[3]:
          Name = Q3
          AxisRef = gAxisQ3
        JointAxis[4]:
          Name = Q4
          AxisRef = gAxisQ4
        JointAxis[5]:
          Name = Q5
          AxisRef = gAxisQ5
    MechanicalSystem:
      MechSysRef = MechSys_5AxRobA
    BasicSettings:
      ModalDataBehaviour = ResetToDefault
      GeometryPlanning:
        TCPResolution:
          LengthResolution = 0.001
          AngleResolution = 0.001
        RoundingMode = Standard
        MaxCornerDeviation = 0.0
        MaxTangentialTransitionDeviation = 0.0
        MaxRadiusDeviation = 0.001
        WorkingPlane = XY
      TrajectoryPlanning = Basic
        LimitCheckResolution = UserDefinedTime
          Time = 0.01
        BufferTime = UserDefinedTime
          Time = 0.1
      Miscellaneous:
        NonMovementsLimit = NotUsed
    AxesGroupFeatures:
      FeatureRef[1] = Feature_Programs
      FeatureRef[2] = Feature_Jogging
      FeatureRef[3] = Feature_Homing
  Alarms = None
```

### Config_2.axis - X20CP0484_1/mappMotion/5AxesRoboarmA/Config_2.axis
```
Element gAxisQ1 (Type=axis)
  BaseTypeIsReadOnly = 0
  BaseType = RotaryBounded
    MeasurementUnitIsReadOnly = 0
    MeasurementUnit = 17476
    MeasurementResolutionIsReadOnly = 0
    MeasurementResolution = 0.01
    CountDirectionIsReadOnly = 0
    CountDirection = Standard
  MovementLimitsIsReadOnly = 0
  MovementLimits = Internal
    Position:
      LowerLimitMin = -1.79769313486231E308
      UpperLimitMax = 1.79769313486231E308
      LowerLimit = -360
      UpperLimit = 360
    VelocityIsReadOnly = 0
    Velocity:
      VelocityMax = 3.4E38
      Velocity = 10.0
    AccelerationIsReadOnly = 0
    Acceleration:
      AccelerationMax = 3.4E38
      Acceleration = 50.0
    DecelerationIsReadOnly = 0
    Deceleration:
      DecelerationMax = 3.4E38
      Deceleration = 50.0
  Alarms = None
Element gAxisQ2 (Type=axis)
  BaseTypeIsReadOnly = 0
  BaseType = RotaryBounded
    MeasurementUnitIsReadOnly = 0
    MeasurementUnit = 17476
    MeasurementResolutionIsReadOnly = 0
    MeasurementResolution = 0.01
    CountDirectionIsReadOnly = 0
    CountDirection = Standard
  MovementLimitsIsReadOnly = 0
  MovementLimits = Internal
    Position:
      LowerLimitMin = -1.79769313486231E308
      UpperLimitMax = 1.79769313486231E308
      LowerLimit = -360
      UpperLimit = 360
    VelocityIsReadOnly = 0
    Velocity:
      VelocityMax = 3.4E38
      Velocity = 10.0
    AccelerationIsReadOnly = 0
    Acceleration:
      AccelerationMax = 3.4E38
      Acceleration = 50.0
    DecelerationIsReadOnly = 0
    Deceleration:
      DecelerationMax = 3.4E38
      Deceleration = 50.0
  Alarms = None
Element gAxisQ3 (Type=axis)
  BaseTypeIsReadOnly = 0
  BaseType = RotaryBounded
    MeasurementUnitIsReadOnly = 0
    MeasurementUnit = 17476
    MeasurementResolutionIsReadOnly = 0
    MeasurementResolution = 0.01
    CountDirectionIsReadOnly = 0
    CountDirection = Standard
  MovementLimitsIsReadOnly = 0
  MovementLimits = Internal
    Position:
      LowerLimitMin = -1.79769313486231E308
      UpperLimitMax = 1.79769313486231E308
      LowerLimit = -360
      UpperLimit = 360
    VelocityIsReadOnly = 0
    Velocity:
      VelocityMax = 3.4E38
      Velocity = 10.0
    AccelerationIsReadOnly = 0
    Acceleration:
      AccelerationMax = 3.4E38
      Acceleration = 50.0
    DecelerationIsReadOnly = 0
    Deceleration:
      DecelerationMax = 3.4E38
      Deceleration = 50.0
  Alarms = None
Element gAxisQ4 (Type=axis)
  BaseTypeIsReadOnly = 0
  BaseType = RotaryBounded
    MeasurementUnitIsReadOnly = 0
    MeasurementUnit = 17476
    MeasurementResolutionIsReadOnly = 0
    MeasurementResolution = 0.01
    CountDirectionIsReadOnly = 0
    CountDirection = Standard
  MovementLimitsIsReadOnly = 0
  MovementLimits = Internal
    Position:
      LowerLimitMin = -1.79769313486231E308
      UpperLimitMax = 1.79769313486231E308
      LowerLimit = -360
      UpperLimit = 360
    VelocityIsReadOnly = 0
    Velocity:
      VelocityMax = 3.4E38
      Velocity = 10.0
    AccelerationIsReadOnly = 0
    Acceleration:
      AccelerationMax = 3.4E38
      Acceleration = 50.0
    DecelerationIsReadOnly = 0
    Deceleration:
      DecelerationMax = 3.4E38
      Deceleration = 50.0
  Alarms = None
Element gAxisQ5 (Type=axis)
  BaseTypeIsReadOnly = 0
  BaseType = RotaryBounded
    MeasurementUnitIsReadOnly = 0
    MeasurementUnit = 17476
    MeasurementResolutionIsReadOnly = 0
    MeasurementResolution = 0.01
    CountDirectionIsReadOnly = 0
    CountDirection = Standard
  MovementLimitsIsReadOnly = 0
  MovementLimits = Internal
    Position:
      LowerLimitMin = -1.79769313486231E308
      UpperLimitMax = 1.79769313486231E308
      LowerLimit = -360
      UpperLimit = 360
    VelocityIsReadOnly = 0
    Velocity:
      VelocityMax = 3.4E38
      Velocity = 10.0
    AccelerationIsReadOnly = 0
    Acceleration:
      AccelerationMax = 3.4E38
      Acceleration = 50.0
    DecelerationIsReadOnly = 0
    Deceleration:
      DecelerationMax = 3.4E38
      Deceleration = 50.0
  Alarms = None
```

### Config_3.mechanicalsystem - X20CP0484_1/mappMotion/5AxesRoboarmA/Config_3.mechanicalsystem
```
Element MechSys_5AxRobA (Type=mechanicalsystem)
  TypeIsReadOnly = 0
  Type = 5AxesRoboarm
    SubtypeIsReadOnly = 0
    Subtype = 5AxesRoboarmA
      DescriptionIsReadOnly = 0
      Description = Standard
        Dimensions:
          TranslationFromBaseToQ1IsReadOnly = 0
          TranslationFromBaseToQ1:
            X = 0.0
            Y = 0.0
            Z = 200
          TranslationFromQ1ToQ2IsReadOnly = 0
          TranslationFromQ1ToQ2:
            X = 0.0
            Y = 0
            Z = 154.5
          TranslationFromQ2ToQ3IsReadOnly = 0
          TranslationFromQ2ToQ3:
            X = 0.0
            Y = 0.0
            Z = 350
          TranslationFromQ3ToQ4IsReadOnly = 0
          TranslationFromQ3ToQ4:
            X = 270
            Y = 0
            Z = 0.0
          TranslationFromQ4ToQ5IsReadOnly = 0
          TranslationFromQ4ToQ5:
            X = 0
            Y = 0
            Z = -190
          TranslationFromQ5ToFlangeIsReadOnly = 0
          TranslationFromQ5ToFlange:
            X = 0.0
            Y = 0.0
            Z = 0
        Offsets:
          JointAxisIsReadOnly = 0
          JointAxis[1] = 0
          JointAxis[2] = -10
          JointAxis[3] = 10
          JointAxis[4] = -60
          JointAxis[5] = -10
        CountDirections:
          JointAxisIsReadOnly = 0
          JointAxis[1] = Inverse
          JointAxis[2] = Inverse
          JointAxis[3] = Inverse
          JointAxis[4] = Inverse
          JointAxis[5] = Inverse
      CoordinatesNames = Default
        XCoordinateName = X
        YCoordinateName = Y
        ZCoordinateName = Z
        BCoordinateName = B
        CCoordinateName = C
      WireFrameModelIsReadOnly = 0
      WireFrameModel = Standard
        Q1ToQ2IsReadOnly = 0
        Q1ToQ2 = ConnectionLine
          DistanceMin = -1.79769313486231E308
          DistanceMax = 1.79769313486231E308
          Distance = 0.0
        Q2ToQ3IsReadOnly = 0
        Q2ToQ3 = ConnectionLine
          DistanceMin = -1.79769313486231E308
          DistanceMax = 1.79769313486231E308
          Distance = 0.0
        Q3ToQ4IsReadOnly = 0
        Q3ToQ4 = ConnectionLine
          DistanceMin = -1.79769313486231E308
          DistanceMax = 1.79769313486231E308
          Distance = 0.0
        Q4ToQ5IsReadOnly = 0
        Q4ToQ5 = ConnectionLine
          DistanceMin = -1.79769313486231E308
          DistanceMax = 1.79769313486231E308
          Distance = 0.0
        Q5ToFlangeIsReadOnly = 0
        Q5ToFlange = ConnectionLine
          DistanceMin = -1.79769313486231E308
          DistanceMax = 1.79769313486231E308
          Distance = 0.0
        FlangeToTcp = ConnectionLine
          DistanceMin = -1.79769313486231E308
          DistanceMax = 1.79769313486231E308
          Distance = 0.0
      DynamicModelIsReadOnly = 0
      DynamicModel = DynParTable
        TableRef
      InternalDynamicModelIsReadOnly = 0
      InternalDynamicModel = NotUsed
      CouplingsIsInvisible = 0
      JointAxesPositionLimits:
        JointAxisIsReadOnly = 0
        JointAxis[1] = UseAxisLimits
        JointAxis[2] = UseAxisLimits
        JointAxis[3] = UseAxisLimits
        JointAxis[4] = UseAxisLimits
        JointAxis[5] = UseAxisLimits
```

### Config_4.axesgroupfeature - X20CP0484_1/mappMotion/5AxesRoboarmA/Config_4.axesgroupfeature
```
Element Feature_Programs (Type=axesgroupfeature)
  Type = Program
    ModalDataBehaviour = UseAxesGroupSettings
    InitialSettings:
      InterpolationTypes = LinearRapid
      PositionCoordinates = Absolute
      CircleCoordinates = Relative
      JACS_ACSProgramming = JACS
      ContourConnection = Inactive
      AccuracyHoldDelays = None
      ProgrammingUnits = UseAxesGroupSettings
      Feedrates:
        FeedPath = Standard
        FeedCharacteristic = StandardCharacteristic
        FeedType = Feedrate
        FeedReduction = Inactive
        FeedrateValue = 0.0
        InverseFeedrateValue = 0.0
        FeedratePerRevValue = 0.0
    DefaultLanguage = BRGCode
    Location = Default
      FileDevice = CNC_PrgDir
Element Feature_Jogging (Type=axesgroupfeature)
  Type = Jogging
Element Feature_Homing (Type=axesgroupfeature)
  Type = HomingOrder
    TogetherGroup[1]:
      AxisRef[1] = gAxisQ1
    TogetherGroup[2]:
      AxisRef[1] = gAxisQ3
      AxisRef[2] = gAxisQ4
      AxisRef[3] = gAxisQ5
      AxisRef[4] = gAxisQ2
Element Feature_Workspace (Type=axesgroupfeature)
  Type = WorkspaceMonitoring
    ModalDataBehaviour = UseAxesGroupSettings
    WorkspaceRef
    SelfCollisionDetection = Enabled
    FlangeWorkspace = NotUsed
```

### Config.mpfilemanager - X20CP0484_1/mappServices/Config.mpfilemanager
```
Element FileManagement (Type=mpfilemanager)
  FileManager:
    Devices:
      0:
        DeviceName = CNC_PrgDir
    Access:
      0:
        Folder = *
        Roles:
          0:
            Role = Everyone
            Rights:
              Visible = TRUE
              FolderRead = TRUE
              FileRead = TRUE
              FileEdit = TRUE
```

### Config_5.mpfilemanagerui - X20CP0484_1/mappServices/Config_5.mpfilemanagerui
```
Element gFileManagerUI (Type=mpfilemanagerui)
```

## Logical view

Binary libraries used (declarations not repeated): operator, runtime, astime, AsIecCon, AsZip, FileIO, AsARCfg, powerlnk, AsEPL, AsIO, sys_lib, DataObj, McBase 5.31.0, MpBase, McPathGen 5.31.0, McAcpAx 5.31.0, McAxis 5.31.0, McStpAx 5.31.0, McProgInt 5.31.0, McAxGroup 5.31.0, MpRobotics 5.31.0, MpAxis 5.31.0, ViBase, CoTrace, McTrkPath 5.31.0, MpPick 5.31.0, AsOpcUac, AsOpcUas

### Global.typ - Global data types
```iecst
TYPE
	VarsHomingSwitchTrigger_typ : 	STRUCT  (*Homing trigger for all axis*)
		Axis1 : BOOL; (*Homing trigger axis 1*)
		Axis2 : BOOL; (*Homing trigger axis 2*)
		Axis3 : BOOL; (*Homing trigger axis 3*)
		Axis4 : BOOL; (*Homing trigger axis 4*)
		Axis5 : BOOL; (*Homing trigger axis 5*)
	END_STRUCT;
	JogDirection_typ : 	STRUCT
		Positive : BOOL;
		Negative : BOOL;
	END_STRUCT;
	GoToState_typ : 	STRUCT  (*Vars from visu*)
		Tipping : BOOL; (*Go to tipping state*)
		GCode : BOOL; (*Go to G-Code state*)
		MoveSetPos : BOOL; (*Go to MoveSetPos state*)
	END_STRUCT;
	HomingCount_enum :
		(
		NoHoming := 0,
		DefaultHomingDone := 1,
		DirectHomingDone := 2
		);
	Pars_typ : 	STRUCT
		PosMCS : ARRAY[0..4]OF LREAL;
	END_STRUCT;
	Cmd_typ : 	STRUCT
		PowerOn : BOOL;
		Home : BOOL;
		Stop : BOOL;
		Start : BOOL;
		ErrorReset : BOOL;
		MoveIndex : BOOL;
	END_STRUCT;
	StateMachine_enum :
		(
		STATE_Disabled := 0,
		STATE_PowerOn := 5,
		STATE_WaitForHome := 9,
		STATE_Home := 10,
		STATE_Idle := 20,
		STATE_Tipping := 40,
		STATE_Error := 99,
		STATE_MoveSetPos := 50
		);
	MainPar_typ : 	STRUCT
		StateMachine : StateMachine_enum;
		PreStateIdent : StateMachine_enum;
		Cmd : Cmd_typ;
		HomingCount : HomingCount_enum;
		Status : Status_enum;
		GoToState : GoToState_typ;
	END_STRUCT;
	Status_enum :
		(
		Disabled,
		Idle,
		State_Active,
		State_Error
		);
END_TYPE
```

### Global.var - Global variables
```iecst
VAR
	gTargetX : LREAL := 0; (*Target TCP X position [mm] from MATLAB*)
	gTargetY : LREAL := 0; (*Target TCP Y position [mm] from MATLAB*)
	gTargetZ : LREAL := 0; (*Target TCP Z position [mm] from MATLAB*)
	gTargetB : LREAL := 0; (*Target TCP B orientation in deg*)
	gTargetC : LREAL := 0; (*Target TCP C orientation in deg*)
	gCmd_MoveLinear : BOOL := FALSE; (*Trigger straight line TCP move*)
	gCmd_Stop : BOOL := FALSE; (*Stop current motion*)
	gCmd_ErrorReset : BOOL := FALSE; (*Reset robot error state*)
	gCmd_MoveDirect : BOOL := FALSE; (*Trigger point to point TCP move*)
	gCmd_JogJoint : BOOL := FALSE; (*Trigger single joint jog step*)
	gJogJointIndex : INT := 0; (*Index of joint to jog*)
	gJogJointStep : LREAL := 0.0; (*Jog step size [deg]*)
	gStatus_Ready : BOOL := FALSE; (*Robot ready to accept commands*)
	gStatus_Moving : BOOL := FALSE; (*Motion currently active*)
	gStatus_InPosition : BOOL := FALSE; (*TCP reached target*)
	gStatus_Error : BOOL := FALSE; (*Error flag*)
	gStatus_ErrorID : DINT := 0; (*Active error code*)
	gStatus_Homed : BOOL := FALSE; (*Robot has been homed*)
	gStatus_PowerOn : BOOL := FALSE; (*Drives powered on*)
	gActual_X : LREAL := 0; (*Live TCP X position [mm]*)
	gActual_Y : LREAL := 0; (*Live TCP Y position [mm]*)
	gActual_Z : LREAL := 0; (*Live TCP Z position [mm]*)
	gActual_B : LREAL := 0; (*Live TCP B orientation [deg]*)
	gActual_C : LREAL := 0; (*Live TCP C orientation [deg]*)
	gActual_Q1 : LREAL := 0; (*Live joint angle Q1 [deg]*)
	gActual_Q2 : LREAL := 0; (*Live joint angle Q2 [deg]*)
	gActual_Q3 : LREAL := 0; (*Live joint angle Q3 [deg]*)
	gActual_Q4 : LREAL := 0; (*Live joint angle Q4 [deg]*)
	gActual_Q5 : LREAL := 0; (*Live joint angle Q5 [deg]*)
	gParam_Velocity : REAL := 10; (*Path velocity limit [mm/s]*)
	gParam_Acceleration : REAL := 50; (*Path acceleration limit [mm/s²]*)
	gParam_Override : REAL := 100; (*Speed override [%]*)
	gEStop_Active : BOOL := FALSE; (*Emergency stop pressed*)
	gEStop_OK : BOOL := TRUE; (*E-stop circuit healthy*)
	RoboParameters : MpRoboArm5AxisParType; (*Parameters for MpRoboArm5Axis*)
	MpRoboArm5Axis_0 : MpRoboArm5Axis; (*Robot motion function block instance*)
	fbMpAxisBasic : ARRAY[0..4] OF MpAxisBasic; (*Single-axis FBs for Q1-Q5*)
	ParAxis : ARRAY[0..4] OF MpAxisBasicParType; (*Per-Axis parameters for Q1-Q5*)
	gAngleOffset_Q1 : LREAL := 0; (*Home offset for Q1 [deg]*)
	gAngleOffset_Q2 : LREAL := -10; (*Home offset for Q2 [deg]*)
	gAngleOffset_Q3 : LREAL := 10; (*Home offset for Q3 [deg]*)
	gAngleOffset_Q4 : LREAL := -60; (*Home offset for Q4 [deg]*)
	gAngleOffset_Q5 : LREAL := -10; (*Home offset for Q1 [deg]*)
	gZeroedAngle_Q1 : LREAL; (*Q1 angle relative to home [deg]*)
	gZeroedAngle_Q2 : LREAL; (*Q2 angle relative to home [deg]*)
	gZeroedAngle_Q3 : LREAL; (*Q3 angle relative to home [deg]*)
	gZeroedAngle_Q4 : LREAL; (*Q4 angle relative to home [deg]*)
	gZeroedAngle_Q5 : LREAL; (*Q5 angle relative to home [deg]*)
	gPickX : LREAL := 0; (*Taught pick position X [mm]*)
	gPickY : LREAL := 0; (*Taught pick position Y [mm]*)
	gPickZ : LREAL := 0; (*Taught pick position Z [mm]*)
	gPickB : LREAL := 0; (*Taught pick orientation B [deg]*)
	gPickC : LREAL := 0; (*Taught pick orientation C [deg]*)
	gPlaceX : LREAL := 0; (*Taught place position X [mm]*)
	gPlaceY : LREAL := 0; (*Taught place position Y [mm]*)
	gPlaceZ : LREAL := 0; (*Taught place position Z [mm]*)
	gPlaceB : LREAL := 0; (*Taught place orientation B [deg]*)
	gPlaceC : LREAL := 0; (*Taught place orientation C [deg]*)
	gHomeX : LREAL := 0; (*Taught home position X [mm]*)
	gHomeY : LREAL := 0; (*Taught home position Y [mm]*)
	gHomeZ : LREAL := 0; (*Taught home position Z [mm]*)
	gHomeB : LREAL := 0; (*Taught home orientation B [deg]*)
	gHomeC : LREAL := 0; (*Taught home orientation C [deg]*)
	PP_OFFSET : LREAL := 80; (*Safe approach height above pick/place [mm]*)
	gCmd_TeachPick : BOOL := FALSE; (*Safe current TCP as pick position*)
	gCmd_TeachPlace : BOOL := FALSE; (*Safe current TCP as place position*)
	gCmd_TeachHome : BOOL := FALSE; (*Safe current TCP as home position*)
	SM_Module_TriggerVars : VarsHomingSwitchTrigger_typ; (*Homing switch trigger signals*)
	gCmd_Home : BOOL; (*Trigger homing sequence from MATLAB HMI*)
	gStatus_Homing : BOOL; (*TRUE while homing is in progress*)
END_VAR
```

### Package Logical/Libraries - Global libraries

### Robotic.st
```iecst
VAR CONSTANT
P099 : McPointType := (Pos:=(X:=280, Y:=0, Z:=525),  Orient:=(Angle1 := -5, Angle2 := 4));
P001 : McPointType := (Pos:=(X:=350, Y:=-60, Z:=500),  Orient:=(Angle1 := -5, Angle2 := 4));
P002 : McPointType := (Pos:=(X:=350, Y:=-60, Z:=400));
P003 : McPointType := (Pos:=(X:=410, Y:=-65, Z:=300));
P004 : McPointType := (Pos:=(X:=350, Y:=-60, Z:=300), Orient:=(Angle1 := -5, Angle2 := 4));
P005 : McPointType := (Pos:=(X:=350, Y:=-60, Z:=500));
P006 : McPointType := (Pos:=(X:=400, Y:=-200, Z:=500));
P007 : McPointType := (Pos:=(X:=450, Y:=-350, Z:=303));
P008 : McPointType := (Pos:=(X:=450, Y:=-350, Z:=400));

END_VAR

	PROGRAM _MAIN

	Feedrate(40 * 40);
	MoveL(P099);//
	MoveL(P001);
	DO_PATH_SYNCH
	GripperClose:= FALSE;
	GripperOpen:= TRUE;
	END_PATH_SYNCH
	MoveL(P002);
	WaitTime(1);
	MoveL(P003);
	DO_PATH_SYNCH
	GripperClose:= TRUE;
	GripperOpen:= FALSE;
	END_PATH_SYNCH
	WaitTime(1);
	MoveL(P004);
	WaitTime(1);
	MoveL(P005);
	MoveL(P006);
	MoveL(P007);
	DO_PATH_SYNCH
	GripperClose:= FALSE;
	GripperOpen:= TRUE;
	END_PATH_SYNCH
	MoveL(P007);
	WaitTime(1);
	MoveL(P008);
	WaitTime(1);
	MoveL(P099);
	END_PROGRAM
```

### Gripper_Open.st
```iecst
VAR{AT 'Program'}

GripperClose: BOOL;
GripperOpen: BOOL;

	END_VAR

	PROGRAM _MAIN

	DO_PATH_SYNCH
	GripperClose:= FALSE;
	GripperOpen:= TRUE;
	END_PATH_SYNCH

	END_PROGRAM
```

### Gripper_Close.st
```iecst
VAR{AT 'Program'}

GripperClose: BOOL;
GripperOpen: BOOL;

	END_VAR

	PROGRAM _MAIN

	DO_PATH_SYNCH
	GripperClose:= TRUE;
	GripperOpen:= FALSE;
	END_PATH_SYNCH

	END_PROGRAM
```

- Visualisation Logical/mappView (not shown)

### Program Logical/Motion_Control (IEC)

#### Variables.var
```iecst
VAR
	initDone : BOOL := FALSE; (*First-Cycle initialization*)
	i : INT; (*loop index*)
	allAxesHomed : BOOL; (*All axes homed*)
	allAxesPowered : BOOL; (*All axes powered*)
	gGripperOpen : BOOL; (*Gripper open*)
	gGripperClose : BOOL; (*Gripper close*)
	pickPlaceStep : INT := 0; (*Current step in the pick and place state machine*)
	gCmd_PickPlace : BOOL := FALSE; (*Start pick and place sequence*)
	ppGripperDelay : INT := 0; (*Cycle counter for gripper settle delay*)
	trigMoveLinear : r_trig; (*Rising-edge trigger for linear move*)
	trigStop : r_trig; (*Rising-edge trigger for stop*)
	trigErrorReset : r_trig; (*Rising-edge trigger for error reset*)
	trigMoveDirect : r_trig; (*Rising-edge trigger for direct move*)
	trigJogJoint : r_trig; (*Rising-edge trigger for joint jog*)
	trigTeachPick : r_trig; (*Rising-edge trigger to teach pick*)
	trigTeachPlace : r_trig; (*Rising-edge trigger to teach place*)
	trigTeachHome : r_trig; (*Rising-edge trigger to teach home*)
	trigHome : r_trig; (*Rising-edge trigger for home*)
	cStandHeight : REAL := 200; (*Stand Height*)
END_VAR
```

#### Main.st
```iecst
(*
================================================================================
  Main.st — Cyclic program for the robot arm
  Hardware : B&R X20CP0484-1 + Igus RL-DP-5
  mapp Motion : 5.22.2  |  Automation Runtime : B4.93

MATLAB sends Cartisian targets (X,Y,Z,B,C) over OPC UA
The PLC handles all kinematics via MpRoboArm5Axis
MpAxisBasic handles per-axis power and homing
================================================================================
*)

PROGRAM _CYCLIC

    // =========================================================================
    // 1. FIRST CYCLE INITIALIZATION
    // =========================================================================
	IF NOT initDone THEN

		// -- Link each axis FB to its configured axis --
		fbMpAxisBasic[0].MpLink     := ADR(gAxisQ1);
		fbMpAxisBasic[1].MpLink     := ADR(gAxisQ2);
		fbMpAxisBasic[2].MpLink     := ADR(gAxisQ3);
		fbMpAxisBasic[3].MpLink     := ADR(gAxisQ4);
		fbMpAxisBasic[4].MpLink     := ADR(gAxisQ5);

		// -- Enable all axes, set default homing --
		FOR i := 0 TO 4 DO
			fbMpAxisBasic[i].Enable     := TRUE;
			fbMpAxisBasic[i].Parameters := ADR(ParAxis[i]);
			ParAxis[i].Velocity         := gParam_Velocity;
			ParAxis[i].Homing.Mode      := mcHOMING_DEFAULT;
		END_FOR;

		// -- MpRoboArm5Axis setup --
		MpRoboArm5Axis_0.MpLink     := ADR(g5AxRobA);
		MpRoboArm5Axis_0.Parameters := ADR(RoboParameters);
		MpRoboArm5Axis_0.Enable     := TRUE;
		MpRoboArm5Axis_0.Override   := 100.0;

		// -- Initialize RoboParameters --
		RoboParameters.CoordSystem    := mcMCS;
		RoboParameters.Velocity     := gParam_Velocity;
		RoboParameters.Acceleration := gParam_Acceleration;
		RoboParameters.Deceleration := gParam_Acceleration;
		RoboParameters.Position[0]  := 0.0;
		RoboParameters.Position[1]  := 0.0;
		RoboParameters.Position[2]  := 0.0;
		RoboParameters.Position[3]  := 0.0;
		RoboParameters.Position[4]  := 0.0;

		// -- Clean command state --
		gCmd_MoveLinear := FALSE;
		gCmd_MoveDirect := FALSE;
		gCmd_Stop       := FALSE;
		gCmd_ErrorReset := FALSE;
		gCmd_Home       := FALSE;

		initDone := TRUE;
	END_IF;

	// =========================================================================
	// 2. ENABLE ALL AXIS BASIC FBs EVERY CYCLE
	// =========================================================================
	FOR i := 0 TO 4 DO
		fbMpAxisBasic[i].Enable := TRUE;
	END_FOR;

	// =========================================================================
	// 3. ENABLE MpRoboArm5Axis EVERY CYCLE
	// =========================================================================
	MpRoboArm5Axis_0.Enable   := TRUE;
	MpRoboArm5Axis_0.Override := gParam_Override;

	// =========================================================================
	// 4. PARAMETER SYNC
	// =========================================================================
	RoboParameters.Velocity     := gParam_Velocity;
	RoboParameters.Acceleration := gParam_Acceleration;
	RoboParameters.Deceleration := gParam_Acceleration;

	FOR i := 0 TO 4 DO
		ParAxis[i].Velocity := gParam_Velocity;
	END_FOR;

	// =========================================================================
	// 5. E-STOP HANDLING
	// =========================================================================
	gEStop_Active := NOT gEStop_OK;

	IF gEStop_Active THEN
		FOR i := 0 TO 4 DO
			fbMpAxisBasic[i].Stop := TRUE;
		END_FOR;
		MpRoboArm5Axis_0.Stop   := TRUE;
		gCmd_MoveLinear         := FALSE;
		gCmd_MoveDirect         := FALSE;
		gCmd_Stop               := FALSE;
	ELSE
		FOR i := 0 TO 4 DO
			fbMpAxisBasic[i].Stop := FALSE;
		END_FOR;
		MpRoboArm5Axis_0.Stop := FALSE;
	END_IF;

	// =========================================================================
	// 6. ERROR RESET
	// =========================================================================
	trigErrorReset(CLK := gCmd_ErrorReset);
	IF trigErrorReset.Q THEN
		FOR i := 0 TO 4 DO
			fbMpAxisBasic[i].ErrorReset := TRUE;
		END_FOR;
		MpRoboArm5Axis_0.ErrorReset := TRUE;
		gCmd_ErrorReset             := FALSE;
	ELSE
		FOR i := 0 TO 4 DO
			IF fbMpAxisBasic[i].ErrorReset AND NOT fbMpAxisBasic[i].Error THEN
				fbMpAxisBasic[i].ErrorReset := FALSE;
			END_IF;
		END_FOR;
		IF MpRoboArm5Axis_0.ErrorReset AND NOT MpRoboArm5Axis_0.Error THEN
			MpRoboArm5Axis_0.ErrorReset := FALSE;
		END_IF;
	END_IF;

	// =========================================================================
	// 6b. HOMING COMMAND — triggered by MATLAB Home button via OPC UA
	// =========================================================================
	trigHome(CLK := gCmd_Home);
	IF trigHome.Q THEN
		gCmd_Home      := FALSE;
		gStatus_Homing := TRUE;
		FOR i := 0 TO 4 DO
			fbMpAxisBasic[i].Home := TRUE;
		END_FOR;
	END_IF;

	// =========================================================================
	// 7. COMMAND PROCESSING — MOVE LINEAR
	// =========================================================================
	trigMoveLinear(CLK := gCmd_MoveLinear);

	IF trigMoveLinear.Q THEN
		gCmd_MoveLinear := FALSE;

		IF gEStop_Active THEN
			// Reject: E-stop

		ELSIF NOT gStatus_Homed THEN
			gStatus_Error   := TRUE;
			gStatus_ErrorID := -1;  // not homed

		ELSIF MpRoboArm5Axis_0.Error THEN
			// Reject: error state

		ELSIF NOT MpRoboArm5Axis_0.PowerOn THEN
			gStatus_Error   := TRUE;
			gStatus_ErrorID := -2;  // power not on

		ELSE
			RoboParameters.Position[0]  := gTargetX;
			RoboParameters.Position[1]  := gTargetY;
			RoboParameters.Position[2]  := gTargetZ;
			RoboParameters.Position[3]  := gTargetB;
			RoboParameters.Position[4]  := gTargetC;

			gStatus_InPosition          := FALSE;
			MpRoboArm5Axis_0.MoveLinear := TRUE;
			MpRoboArm5Axis_0.MoveDirect := FALSE;
		END_IF;
	END_IF;

	// =========================================================================
	// 8. COMMAND PROCESSING — MOVE DIRECT
	// =========================================================================
	trigMoveDirect(CLK := gCmd_MoveDirect);

	IF trigMoveDirect.Q THEN
		gCmd_MoveDirect := FALSE;

		IF gEStop_Active THEN
			// Reject

		ELSIF NOT gStatus_Homed THEN
			gStatus_Error   := TRUE;
			gStatus_ErrorID := -1;

		ELSIF MpRoboArm5Axis_0.Error THEN
			// Reject

		ELSIF NOT MpRoboArm5Axis_0.PowerOn THEN
			gStatus_Error   := TRUE;
			gStatus_ErrorID := -2;

		ELSE
			RoboParameters.Position[0]  := gTargetX;
			RoboParameters.Position[1]  := gTargetY;
			RoboParameters.Position[2]  := gTargetZ;
			RoboParameters.Position[3]  := gTargetB;
			RoboParameters.Position[4]  := gTargetC;

			gStatus_InPosition          := FALSE;
			MpRoboArm5Axis_0.MoveDirect := TRUE;
			MpRoboArm5Axis_0.MoveLinear := FALSE;
		END_IF;
	END_IF;

	// =========================================================================
	// 8b. COMMAND PROCESSING — JOINT JOG (ACS — single joint only)
	// =========================================================================
	trigJogJoint(CLK := gCmd_JogJoint);
	IF trigJogJoint.Q THEN
		gCmd_JogJoint := FALSE;

		IF NOT gEStop_Active AND NOT MpRoboArm5Axis_0.Error
			AND gStatus_PowerOn AND gStatus_Homed THEN

			RoboParameters.CoordSystem := mcACS;

			RoboParameters.Position[0] := MpRoboArm5Axis_0.Info.JointAxisPosition[0];
			RoboParameters.Position[1] := MpRoboArm5Axis_0.Info.JointAxisPosition[1];
			RoboParameters.Position[2] := MpRoboArm5Axis_0.Info.JointAxisPosition[2];
			RoboParameters.Position[3] := MpRoboArm5Axis_0.Info.JointAxisPosition[3];
			RoboParameters.Position[4] := MpRoboArm5Axis_0.Info.JointAxisPosition[4];

			CASE gJogJointIndex OF
				1: RoboParameters.Position[0] := RoboParameters.Position[0] + gJogJointStep;
				2: RoboParameters.Position[1] := RoboParameters.Position[1] + gJogJointStep;
				3: RoboParameters.Position[2] := RoboParameters.Position[2] + gJogJointStep;
				4: RoboParameters.Position[3] := RoboParameters.Position[3] + gJogJointStep;
				5: RoboParameters.Position[4] := RoboParameters.Position[4] + gJogJointStep;
			END_CASE;

			gStatus_InPosition          := FALSE;
			MpRoboArm5Axis_0.MoveLinear := FALSE;
			MpRoboArm5Axis_0.MoveDirect := TRUE;
		END_IF;
	END_IF;

	// =========================================================================
	// 9. COMMAND PROCESSING — STOP
	// =========================================================================
	trigStop(CLK := gCmd_Stop);
	IF trigStop.Q THEN
		gCmd_Stop                   := FALSE;
		MpRoboArm5Axis_0.MoveLinear := FALSE;
		MpRoboArm5Axis_0.MoveDirect := FALSE;
		MpRoboArm5Axis_0.Stop       := TRUE;
	END_IF;

	IF MpRoboArm5Axis_0.Stop AND NOT gEStop_Active THEN
		MpRoboArm5Axis_0.Stop := FALSE;
	END_IF;

	// =========================================================================
	// 10. MOVE COMPLETION DETECTION
	// =========================================================================
	IF MpRoboArm5Axis_0.MoveLinear OR MpRoboArm5Axis_0.MoveDirect THEN
		IF MpRoboArm5Axis_0.MoveDone THEN
			MpRoboArm5Axis_0.MoveLinear := FALSE;
			MpRoboArm5Axis_0.MoveDirect := FALSE;
			gStatus_InPosition          := TRUE;
			gStatus_Moving              := FALSE;
		ELSIF MpRoboArm5Axis_0.Error OR MpRoboArm5Axis_0.CommandAborted THEN
			MpRoboArm5Axis_0.MoveLinear := FALSE;
			MpRoboArm5Axis_0.MoveDirect := FALSE;
			gStatus_Moving              := FALSE;
		ELSE
			gStatus_Moving     := TRUE;
			gStatus_InPosition := FALSE;
		END_IF;
	END_IF;

	RoboParameters.CoordSystem := mcMCS;

	// =========================================================================
	// 11. CALL MpAxisBasic FOR ALL 5 JOINTS EVERY CYCLE
	// =========================================================================
	FOR i := 0 TO 4 DO
		fbMpAxisBasic[i]();
	END_FOR;

	// =========================================================================
	// 12. CALL MpRoboArm5Axis EVERY CYCLE
	// =========================================================================
	MpRoboArm5Axis_0();

	// =========================================================================
	// 13. STATUS OUTPUT PUBLISHING
	// =========================================================================
	allAxesHomed := fbMpAxisBasic[0].IsHomed AND fbMpAxisBasic[1].IsHomed
	AND fbMpAxisBasic[2].IsHomed AND fbMpAxisBasic[3].IsHomed
	AND fbMpAxisBasic[4].IsHomed;

	allAxesPowered := fbMpAxisBasic[0].PowerOn AND fbMpAxisBasic[1].PowerOn
	AND fbMpAxisBasic[2].PowerOn AND fbMpAxisBasic[3].PowerOn
	AND fbMpAxisBasic[4].PowerOn;

	gStatus_Homed   := MpRoboArm5Axis_0.IsHomed AND allAxesHomed;
	gStatus_PowerOn := MpRoboArm5Axis_0.PowerOn AND allAxesPowered;
	gStatus_Ready   := gStatus_PowerOn AND gStatus_Homed
	AND NOT MpRoboArm5Axis_0.Error;

	IF MpRoboArm5Axis_0.Error THEN
		gStatus_Error   := TRUE;
		gStatus_ErrorID := MpRoboArm5Axis_0.StatusID;
	ELSIF NOT gEStop_Active THEN
		gStatus_Error   := FALSE;
		gStatus_ErrorID := 0;
	END_IF;

	// Clear Home trigger once all axes finish homing
	IF gStatus_Homing AND allAxesHomed THEN
		FOR i := 0 TO 4 DO
			fbMpAxisBasic[i].Home := FALSE;
		END_FOR;
		gStatus_Homing := FALSE;
	END_IF;

	// =========================================================================
	// 14. ACTUAL POSITION FEEDBACK
	// =========================================================================
	gActual_X := MpRoboArm5Axis_0.X;
	gActual_Y := MpRoboArm5Axis_0.Y;
	gActual_Z := MpRoboArm5Axis_0.Z;
	gActual_B := MpRoboArm5Axis_0.B;
	gActual_C := MpRoboArm5Axis_0.C;

	gActual_Q1 := MpRoboArm5Axis_0.Info.JointAxisPosition[0];
	gActual_Q2 := MpRoboArm5Axis_0.Info.JointAxisPosition[1];
	gActual_Q3 := MpRoboArm5Axis_0.Info.JointAxisPosition[2];
	gActual_Q4 := MpRoboArm5Axis_0.Info.JointAxisPosition[3];
	gActual_Q5 := MpRoboArm5Axis_0.Info.JointAxisPosition[4];

	gZeroedAngle_Q1 := -(gActual_Q1 - gAngleOffset_Q1);
	gZeroedAngle_Q2 := -(gActual_Q2 - gAngleOffset_Q2);
	gZeroedAngle_Q3 := -(gActual_Q3 - gAngleOffset_Q3);
	gZeroedAngle_Q4 := -(gActual_Q4 - gAngleOffset_Q4);
	gZeroedAngle_Q5 := -(gActual_Q5 - gAngleOffset_Q5);

	// =========================================================================
	// 15. TEACH POSITIONS — store actual TCP into pick/place/home variables
	// =========================================================================
	trigTeachPick(CLK := gCmd_TeachPick);
	IF trigTeachPick.Q THEN
		gCmd_TeachPick := FALSE;
		gPickX := MpRoboArm5Axis_0.X;
		gPickY := MpRoboArm5Axis_0.Y;
		gPickZ := MpRoboArm5Axis_0.Z;
		gPickB := MpRoboArm5Axis_0.B;
		gPickC := MpRoboArm5Axis_0.C;
	END_IF;

	trigTeachPlace(CLK := gCmd_TeachPlace);
	IF trigTeachPlace.Q THEN
		gCmd_TeachPlace := FALSE;
		gPlaceX := MpRoboArm5Axis_0.X;
		gPlaceY := MpRoboArm5Axis_0.Y;
		gPlaceZ := MpRoboArm5Axis_0.Z;
		gPlaceB := MpRoboArm5Axis_0.B;
		gPlaceC := MpRoboArm5Axis_0.C;
	END_IF;

	trigTeachHome(CLK := gCmd_TeachHome);
	IF trigTeachHome.Q THEN
		gCmd_TeachHome := FALSE;
		gHomeX := MpRoboArm5Axis_0.X;
		gHomeY := MpRoboArm5Axis_0.Y;
		gHomeZ := MpRoboArm5Axis_0.Z;
		gHomeB := MpRoboArm5Axis_0.B;
		gHomeC := MpRoboArm5Axis_0.C;
	END_IF;

	// =========================================================================
	// 16. PICK AND PLACE : Home --> above Pick --> Pick --> grip --> above Pick --> above Place --> Place --> release --> above Place --> Home
	//     PP_OFFSET      : safe height above pick / place
	//     ppGripperDelay : wait counter for gripper to settle (~300 cycles)
	// =========================================================================
	IF gCmd_PickPlace THEN
		CASE pickPlaceStep OF

			0:  // Start at home — open gripper
				gTargetX        := gHomeX;
				gTargetY        := gHomeY;
				gTargetZ        := gHomeZ;
				gTargetB        := gHomeB;
				gTargetC        := gHomeC;
				gCmd_MoveDirect := TRUE;
				gGripperOpen    := TRUE;
				gGripperClose   := FALSE;
				pickPlaceStep   := 1;

			1:  // Wait at home
				IF gStatus_InPosition THEN
					ppGripperDelay := ppGripperDelay + 1;
					IF ppGripperDelay >= 300 THEN
						ppGripperDelay := 0;
						pickPlaceStep  := 2;
					END_IF;
				END_IF;

			2:  // Move above pick point
				gTargetX        := gPickX;
				gTargetY        := gPickY;
				gTargetZ        := gPickZ + PP_OFFSET;
				gTargetB        := gPickB;
				gTargetC        := gPickC;
				gCmd_MoveDirect := TRUE;
				pickPlaceStep   := 3;

			3:  // Wait above pick
				IF gStatus_InPosition THEN
					pickPlaceStep := 4;
				END_IF;

			4:  // Lower straight down to pick point
				gTargetX        := gPickX;
				gTargetY        := gPickY;
				gTargetZ        := gPickZ;
				gTargetB        := gPickB;
				gTargetC        := gPickC;
				gCmd_MoveLinear := TRUE;
				pickPlaceStep   := 5;

			5:  // Wait at pick point
				IF gStatus_InPosition THEN
					pickPlaceStep := 6;
				END_IF;

			6:  // Close gripper — grip object
				gGripperClose     := TRUE;
				gGripperOpen      := FALSE;
				ppGripperDelay    := ppGripperDelay + 1;
				IF ppGripperDelay >= 300 THEN
					ppGripperDelay := 0;
					pickPlaceStep  := 7;
				END_IF;

			7:  // Lift straight up above pick
				gTargetX        := gPickX;
				gTargetY        := gPickY;
				gTargetZ        := gPickZ + PP_OFFSET;
				gTargetB        := gPickB;
				gTargetC        := gPickC;
				gCmd_MoveLinear := TRUE;
				pickPlaceStep   := 8;

			8:  // Wait above pick
				IF gStatus_InPosition THEN
					pickPlaceStep := 9;
				END_IF;

			9:  // Move across to above place point
				gTargetX        := gPlaceX;
				gTargetY        := gPlaceY;
				gTargetZ        := gPlaceZ + PP_OFFSET;
				gTargetB        := gPlaceB;
				gTargetC        := gPlaceC;
				gCmd_MoveDirect := TRUE;
				pickPlaceStep   := 10;

			10: // Wait above place
				IF gStatus_InPosition THEN
					pickPlaceStep := 11;
				END_IF;

			11: // Lower straight down to place point
				gTargetX        := gPlaceX;
				gTargetY        := gPlaceY;
				gTargetZ        := gPlaceZ;
				gTargetB        := gPlaceB;
				gTargetC        := gPlaceC;
				gCmd_MoveLinear := TRUE;
				pickPlaceStep   := 12;

			12: // Wait at place point
				IF gStatus_InPosition THEN
					pickPlaceStep := 13;
				END_IF;

			13: // Open gripper — release object
				gGripperOpen      := TRUE;
				gGripperClose     := FALSE;
				ppGripperDelay    := ppGripperDelay + 1;
				IF ppGripperDelay >= 300 THEN
					ppGripperDelay := 0;
					pickPlaceStep  := 14;
				END_IF;

			14: // Lift above place point
				gTargetX        := gPlaceX;
				gTargetY        := gPlaceY;
				gTargetZ        := gPlaceZ + PP_OFFSET;
				gTargetB        := gPlaceB;
				gTargetC        := gPlaceC;
				gCmd_MoveLinear := TRUE;
				pickPlaceStep   := 15;

			15: // Wait above place
				IF gStatus_InPosition THEN
					pickPlaceStep := 16;
				END_IF;

			16: // Return to home
				gTargetX        := gHomeX;
				gTargetY        := gHomeY;
				gTargetZ        := gHomeZ;
				gTargetB        := gHomeB;
				gTargetC        := gHomeC;
				gCmd_MoveDirect := TRUE;
				pickPlaceStep   := 17;

			17: // Wait at home — sequence complete
				IF gStatus_InPosition THEN
					gGripperOpen   := FALSE;
					gGripperClose  := FALSE;
					gCmd_PickPlace := FALSE;
					pickPlaceStep  := 0;
				END_IF;

		END_CASE;
	END_IF;

END_PROGRAM
```
